FUNCTION_BLOCK FB_BA_AdsComClient EXTENDS FB_BA_VIEW
VAR_INPUT
END_VAR
VAR_OUTPUT
END_VAR
VAR_INPUT CONSTANT
	WeatherStation					: FB_BA_RawSubscriber;
	WeatherStationError				: FB_BA_BV;											

	GeneralSettings					: FB_BA_RawSubscriber;												
	GeneralSettingsError			: FB_BA_BV;			
END_VAR
VAR
END_VAR

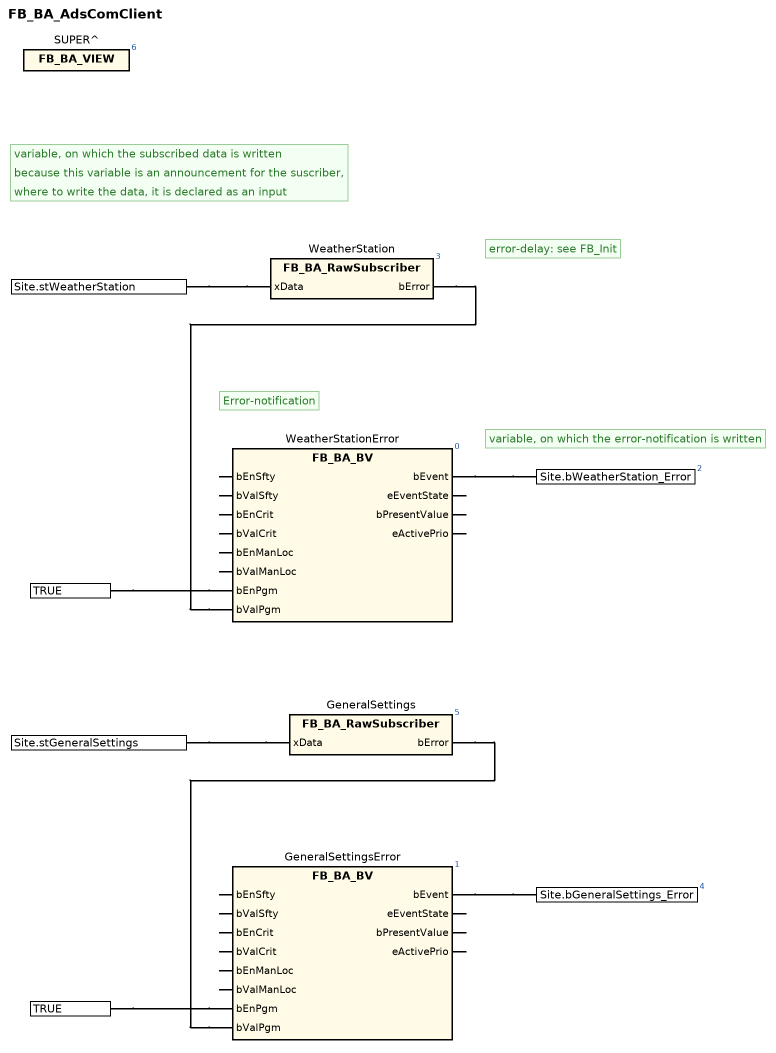
// Error-notification
WeatherStationError(bEnPgm := TRUE, bValPgm := WeatherStation.bError); // FB_BA_BV
GeneralSettingsError(bEnPgm := TRUE, bValPgm := GeneralSettings.bError); // FB_BA_BV
// variable, on which the error-notification is written
Site.bWeatherStation_Error := WeatherStationError.bEvent;
// variable, on which the subscribed data is written
// because this variable is an announcement for the suscriber,
// where to write the data, it is declared as an input
// error-delay: see FB_Init
WeatherStation(xData := Site.stWeatherStation); // FB_BA_RawSubscriber
Site.bGeneralSettings_Error := GeneralSettingsError.bEvent;
GeneralSettings(xData := Site.stGeneralSettings); // FB_BA_RawSubscriber
SUPER^(); // FB_BA_VIEW

METHOD FB_init : BOOL
VAR_INPUT
	bInitRetains : BOOL; // if TRUE, the retain variables are initialized (warm start / cold start)
	bInCopyCode : BOOL;  // if TRUE, the instance afterwards gets moved into the copy code (online change)
END_VAR
WeatherStation.Subject							:= Site.WeatherStation_Subject;		// instance-name of the publisher in the source
WeatherStation.sTarget							:= Site.WeatherStation_NetId;		// AMS-Net-Id of the publishing controller
WeatherStation.tReadInterval					:= T#5S;							// subscribe-interval
WeatherStation.tReadTolerance					:= T#60S;							// delay time, until an erroneous communication will be displayed at the error-output of the subscriber

WeatherStationError.iParent						:= THIS^;
WeatherStationError.iLabel						:= LblAgg_WeatherStationComm;
WeatherStationError.sActiveText 				:= txtEvent_Triggered;
WeatherStationError.sInactiveText 				:= txtEvent_Normal;
WeatherStationError.bEnManualRm					:= FALSE;	//	Priority  8	
WeatherStationError.bValManualRm				:= FALSE;	//	Priority  8
WeatherStationError.nEventClassID				:= EC_ID.NC30;
WeatherStationError.stTimeDelay.nToNormal		:= 0;
WeatherStationError.stTimeDelay.nToAbnormal		:= 0;
WeatherStationError.bAlarmValue					:= TRUE;
WeatherStationError.aEventTransitionText[1]		:= txtEvent_Disturb;
WeatherStationError.aEventTransitionText[2]		:= txtEvent_None;
WeatherStationError.aEventTransitionText[3]		:= txtEvent_Normal;
WeatherStationError.bEventDetectionEnable		:= TRUE;
WeatherStationError.eEnPlantLock				:= E_BA_LockPriority.eNoLock;

GeneralSettings.Subject							:= Site.GeneralSettings_Subject;	// instance-name of the publisher in the source
GeneralSettings.sTarget							:= Site.GeneralSettings_NetId;		// AMS-Net-Id of the publishing controller
GeneralSettings.tReadInterval					:= T#5S;							// subscribe-interval
GeneralSettings.tReadTolerance					:= T#60S;							// delay time, until an erroneous communication will be displayed at the error-output of the subscriber

GeneralSettingsError.iParent					:= THIS^;
GeneralSettingsError.iLabel						:= LblAgg_GeneralSettingsCom;
//GeneralSettingsError.sObjectName				:= F_BA_CONCAT06(s01:= Seperator.sAgg_ObjName, s02:= Agg_GeneralSettingsCom_ObjName, s03:= '02', s04:= Seperator.sFun_ObjName, s05:= Fun_Fault_ObjName, s06:= '01');  
//GeneralSettingsError.sDescription				:= F_BA_CONCAT06(s01:= Seperator.sAgg_Descr, s02:= Agg_GeneralSettingsCom_Descr, s03:= '', s04:= Seperator.sFun_Descr, s05:= Fun_Fault_Descr, s06:= ''); 	
GeneralSettingsError.sActiveText 				:= txtEvent_Triggered;
GeneralSettingsError.sInactiveText 				:= txtEvent_Normal;
GeneralSettingsError.bEnManualRm				:= FALSE;	//	Priority  8	
GeneralSettingsError.bValManualRm				:= FALSE;	//	Priority  8
GeneralSettingsError.nEventClassID				:= EC_ID.NC30;
GeneralSettingsError.stTimeDelay.nToNormal		:= 0;
GeneralSettingsError.stTimeDelay.nToAbnormal	:= 0;
GeneralSettingsError.bAlarmValue				:= TRUE;
GeneralSettingsError.aEventTransitionText[1]	:= txtEvent_Disturb;
GeneralSettingsError.aEventTransitionText[2]	:= txtEvent_None;
GeneralSettingsError.aEventTransitionText[3]	:= txtEvent_Normal;
GeneralSettingsError.bEventDetectionEnable		:= TRUE;
GeneralSettingsError.eEnPlantLock				:= E_BA_LockPriority.eNoLock;
END_METHOD

END_FUNCTION_BLOCK

(* stored: Version 1.1.0.1, ProductVersion 3.1.4024.12
   POU FB_BA_AdsComClient: Id {dbbb7c2f-66eb-4b9b-a5fb-cbeec52577c4}, SpecialFunc None
   Method FB_init: Id {a8cf0598-961f-4b9a-8302-bb285fbe93ef} *)
